FUNCTION_BLOCK Automatik_Betrieb
VAR_INPUT
	Kein_Notaus : BOOL;
	Zyklus_Start : BOOL;
	Zyklus_Stopp : BOOL;
	SFCInit : BOOL;
	SFCTip : BOOL;
	SFCTipMode : BOOL;
	Einfache_Klemmung : BOOL;
	
	//Eingänge Sensorik
	//Zuführer
	Endl_Zufuehrer_Hinten : BOOL;
	Endl_Zufuehrer_Vorne : BOOL;
	Vorposition_Zufuehrer : BOOL;
	IOL_Schaltausg_Distanzsensor_Holzende : BOOL; //Über Schaltausgang oder IO-Link Analogdaten?
	IOL_DistanzSensor_Abst : UINT;
	//Stammklemmung Oben
	Endl_Obere_Stammklemmung_Oben : BOOL;
	Endl_Obere_Stammklemmung_Unten : BOOL;
	Endl_Tastschiene : BOOL;
	Schaltausg_Druckschalter_Obere_Klemmung : BOOL;
	//Stammklemmung Unten
	Endl_Untere_Stammklemmung_Oben : BOOL;
	Endl_Untere_Stammklemmung_Unten : BOOL;
	//Säge
	Endl_Saege_Oben : BOOL;
	Endl_Saege_Unten : BOOL;
	
END_VAR
VAR_OUTPUT
	Warten_Auf_Weiterschalten :BOOL;
	Warten_auf_Material : BOOL;
	//Hydraulik
	QStammklemmung_Oben_Hoch : BOOL;
	QStammklemmung_Oben_Runter : BOOL;
	QStammklemmung_Unten_Hoch : BOOL;
	QStammklemmung_Unten_Runter : BOOL;
	QSaege_Senken : BOOL;
	QSaege_Heben : BOOL;
	//Ausgänge Schalten
	QHydraulikpumpe_EIN : BOOL;
	QZufuehrer_Antrieb_vor : BOOL;
	QZufuehrer_Antrieb_Rueck : BOOL;
	QSaege_Antrieb_Ein : BOOL;
	QKettenschmierung_EIN : BOOL;
	
END_VAR
VAR_IN_OUT
	warten : BOOL;
	Hydraulik_EIN : BOOL;
	Zyklus_Beendet : BOOL;
END_VAR
VAR
	Holz_Fertig : BOOL;
	Holz_Geklemmt : BOOL;
END_VAR

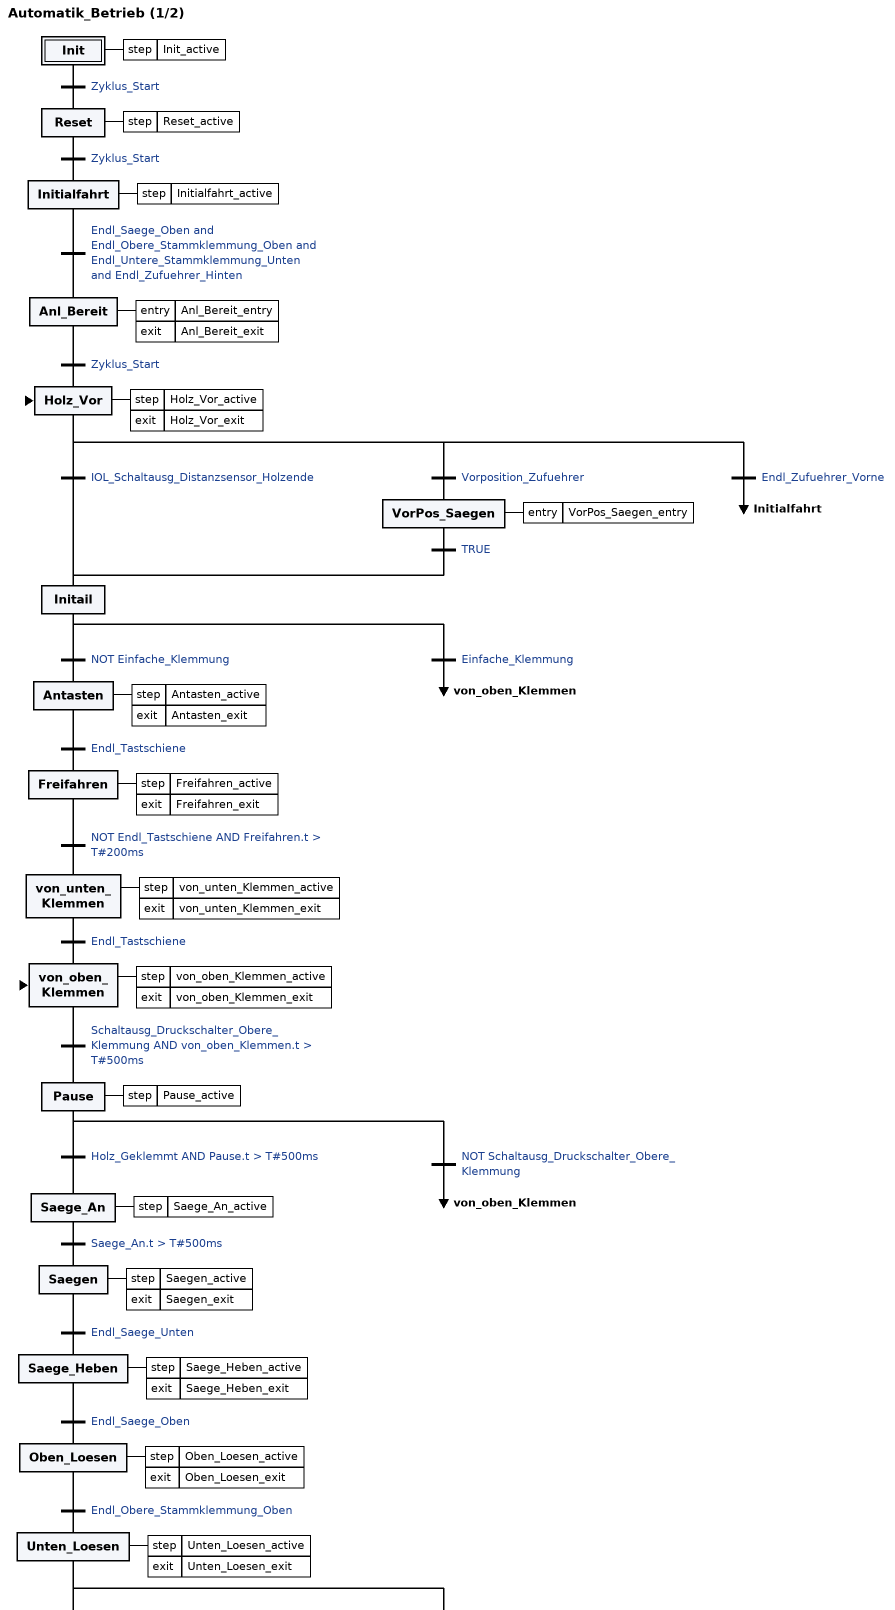
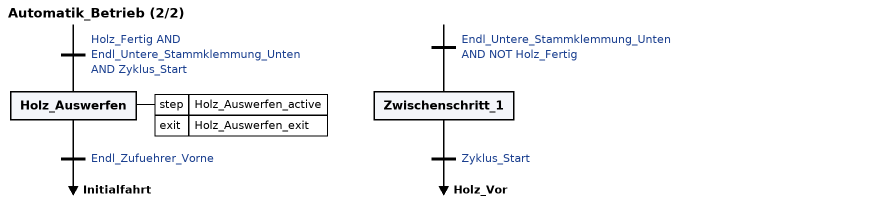
INITIAL_STEP Init:
    Init_active(N);  // step action
END_STEP
TRANSITION FROM Init TO Reset
    := Zyklus_Start;
END_TRANSITION
STEP Reset:
    Reset_active(N);  // step action
END_STEP
TRANSITION FROM Reset TO Initialfahrt_
    := Zyklus_Start;
END_TRANSITION
STEP Initialfahrt_:  // name as stored: Initialfahrt 
    Initialfahrt_active(N);  // step action
END_STEP
TRANSITION FROM Initialfahrt_ TO Anl_Bereit
    := Endl_Saege_Oben and Endl_Obere_Stammklemmung_Oben and Endl_Untere_Stammklemmung_Unten and Endl_Zufuehrer_Hinten;
END_TRANSITION
STEP Anl_Bereit:
    Anl_Bereit_entry(P1);  // entry action
    Anl_Bereit_exit(P0);  // exit action
END_STEP
TRANSITION FROM Anl_Bereit TO Holz_Vor
    := Zyklus_Start;
END_TRANSITION
STEP Holz_Vor:
    Holz_Vor_active(N);  // step action
    Holz_Vor_exit(P0);  // exit action
END_STEP
TRANSITION FROM Holz_Vor TO Initail
    := IOL_Schaltausg_Distanzsensor_Holzende;
END_TRANSITION
TRANSITION FROM Holz_Vor TO VorPos_Saegen
    := Vorposition_Zufuehrer;
END_TRANSITION
STEP VorPos_Saegen:
    VorPos_Saegen_entry(P1);  // entry action
END_STEP
TRANSITION FROM VorPos_Saegen TO Initail
    := TRUE;
END_TRANSITION
TRANSITION FROM Holz_Vor TO Initialfahrt
    := Endl_Zufuehrer_Vorne;
END_TRANSITION
// macro Holz_Klemmen begins
STEP Initail:
END_STEP
TRANSITION FROM Initail TO Antasten
    := NOT Einfache_Klemmung;
END_TRANSITION
STEP Antasten:
    Antasten_active(N);  // step action
    Antasten_exit(P0);  // exit action
END_STEP
TRANSITION FROM Initail TO von_oben_Klemmen
    := Einfache_Klemmung;
END_TRANSITION
TRANSITION FROM Antasten TO Freifahren
    := Endl_Tastschiene;
END_TRANSITION
STEP Freifahren:
    Freifahren_active(N);  // step action
    Freifahren_exit(P0);  // exit action
END_STEP
TRANSITION FROM Freifahren TO von_unten_Klemmen
    := NOT Endl_Tastschiene AND Freifahren.t > T#200ms;
END_TRANSITION
STEP von_unten_Klemmen:
    von_unten_Klemmen_active(N);  // step action
    von_unten_Klemmen_exit(P0);  // exit action
END_STEP
TRANSITION FROM von_unten_Klemmen TO von_oben_Klemmen
    := Endl_Tastschiene;
END_TRANSITION
STEP von_oben_Klemmen:
    von_oben_Klemmen_active(N);  // step action
    von_oben_Klemmen_exit(P0);  // exit action
END_STEP
TRANSITION FROM von_oben_Klemmen TO Pause
    := Schaltausg_Druckschalter_Obere_Klemmung AND von_oben_Klemmen.t > T#500ms;
END_TRANSITION
STEP Pause:
    Pause_active(N);  // step action
END_STEP
TRANSITION FROM Pause TO Saege_An
    := Holz_Geklemmt AND Pause.t > T#500ms;
END_TRANSITION
TRANSITION FROM Pause TO von_oben_Klemmen
    := NOT Schaltausg_Druckschalter_Obere_Klemmung;
END_TRANSITION
// macro Holz_Saegen begins
STEP Saege_An:
    Saege_An_active(N);  // step action
END_STEP
TRANSITION FROM Saege_An TO Saegen
    := Saege_An.t > T#500ms;
END_TRANSITION
STEP Saegen:
    Saegen_active(N);  // step action
    Saegen_exit(P0);  // exit action
END_STEP
TRANSITION FROM Saegen TO Saege_Heben
    := Endl_Saege_Unten;
END_TRANSITION
STEP Saege_Heben:
    Saege_Heben_active(N);  // step action
    Saege_Heben_exit(P0);  // exit action
END_STEP
TRANSITION FROM Saege_Heben TO Oben_Loesen
    := Endl_Saege_Oben;
END_TRANSITION
// macro Holz_Klemmung_Loesen begins
STEP Oben_Loesen:
    Oben_Loesen_active(N);  // step action
    Oben_Loesen_exit(P0);  // exit action
END_STEP
TRANSITION FROM Oben_Loesen TO Unten_Loesen
    := Endl_Obere_Stammklemmung_Oben;
END_TRANSITION
STEP Unten_Loesen:
    Unten_Loesen_active(N);  // step action
    Unten_Loesen_exit(P0);  // exit action
END_STEP
TRANSITION FROM Unten_Loesen TO Holz_Auswerfen
    := Holz_Fertig AND Endl_Untere_Stammklemmung_Unten AND Zyklus_Start;
END_TRANSITION
STEP Holz_Auswerfen:
    Holz_Auswerfen_active(N);  // step action
    Holz_Auswerfen_exit(P0);  // exit action
END_STEP
TRANSITION FROM Holz_Auswerfen TO Initialfahrt
    := Endl_Zufuehrer_Vorne;
END_TRANSITION
TRANSITION FROM Unten_Loesen TO Zwischenschritt_1
    := Endl_Untere_Stammklemmung_Unten AND NOT Holz_Fertig;
END_TRANSITION
STEP Zwischenschritt_1:
END_STEP
TRANSITION FROM Zwischenschritt_1 TO Holz_Vor
    := Zyklus_Start;
END_TRANSITION

ACTION Anl_Bereit_entry:
Warten_auf_Material := TRUE;
QHydraulikpumpe_EIN := FALSE;
END_ACTION

ACTION Anl_Bereit_exit:
Warten_auf_Material := FALSE;
QHydraulikpumpe_EIN := TRUE;
END_ACTION

ACTION Antasten_active:
QStammklemmung_Oben_Runter := TRUE;
END_ACTION

ACTION Antasten_exit:
QStammklemmung_Oben_Runter := FALSE;
END_ACTION

ACTION Freifahren_active:
QStammklemmung_Oben_Hoch := TRUE;
END_ACTION

ACTION Freifahren_exit:
QStammklemmung_Oben_Hoch := FALSE;
END_ACTION

ACTION Holz_Auswerfen_active:
QZufuehrer_Antrieb_vor := TRUE;
END_ACTION

ACTION Holz_Auswerfen_exit:
QZufuehrer_Antrieb_vor := FALSE;
Holz_Fertig := FALSE;
END_ACTION

ACTION Holz_Vor_active:
IF NOT Vorposition_Zufuehrer AND NOT Endl_Zufuehrer_Vorne THEN
	QZufuehrer_Antrieb_vor := TRUE;
END_IF 


IF Vorposition_Zufuehrer OR Endl_Zufuehrer_Vorne OR IOL_Schaltausg_Distanzsensor_Holzende THEN
	QZufuehrer_Antrieb_vor := FALSE;
END_IF
END_ACTION

ACTION Holz_Vor_exit:
QZufuehrer_Antrieb_vor := FALSE;
END_ACTION

ACTION Init_active:
QStammklemmung_Oben_Hoch := 
QStammklemmung_Oben_Runter := 
QStammklemmung_Unten_Hoch := 
QStammklemmung_Unten_Runter := 
QSaege_Senken := 
QSaege_Heben := 
//Ausgänge Schalten
QHydraulikpumpe_EIN := 
QZufuehrer_Antrieb_vor := 
QZufuehrer_Antrieb_Rueck := 
QSaege_Antrieb_Ein := 
QKettenschmierung_EIN := 
Warten_Auf_Weiterschalten :=
Zyklus_Beendet := FALSE;
END_ACTION

ACTION Initialfahrt_active:
IF NOT Endl_Saege_Oben THEN
	QSaege_Heben := TRUE;
	warten := TRUE;
ELSE 
	QSaege_Heben := FALSE;
	warten := FALSE;
END_IF

IF NOT Endl_Obere_Stammklemmung_Oben AND NOT warten THEN
	QStammklemmung_Oben_Hoch := TRUE;
	warten := TRUE;
ELSE
	QStammklemmung_Oben_Hoch := FALSE;
	warten := FALSE;
END_IF

IF NOT Endl_Untere_Stammklemmung_Unten AND NOT warten THEN 
	QStammklemmung_Unten_Runter := TRUE;
	warten := TRUE;
ELSE 
	QStammklemmung_Unten_Runter := FALSE;
	warten := FALSE;
END_IF

IF NOT Endl_Zufuehrer_Hinten THEN
	QZufuehrer_Antrieb_Rueck := TRUE;
ELSE 
	QZufuehrer_Antrieb_Rueck := FALSE;
END_IF
END_ACTION

ACTION Oben_Loesen_active:
QStammklemmung_Oben_Hoch := TRUE;
END_ACTION

ACTION Oben_Loesen_exit:
QStammklemmung_Oben_Hoch := FALSE;
END_ACTION

ACTION Pause_active:
Holz_Geklemmt := TRUE;
END_ACTION

ACTION Reset_active:
//Hydraulik
QStammklemmung_Oben_Hoch := 
QStammklemmung_Oben_Runter := 
QStammklemmung_Unten_Hoch := 
QStammklemmung_Unten_Runter := 
QSaege_Senken := 
QSaege_Heben := 
//Ausgänge Schalten
QHydraulikpumpe_EIN := 
QZufuehrer_Antrieb_vor := 
QZufuehrer_Antrieb_Rueck := 
QSaege_Antrieb_Ein := 
QKettenschmierung_EIN := 
Warten_Auf_Weiterschalten :=
Zyklus_Beendet := FALSE;

QHydraulikpumpe_EIN := TRUE;
END_ACTION

ACTION Saege_An_active:
QSaege_Antrieb_Ein := TRUE;
END_ACTION

ACTION Saege_Heben_active:
QSaege_Heben := TRUE;
END_ACTION

ACTION Saege_Heben_exit:
QSaege_Heben := FALSE;
QSaege_Antrieb_Ein := FALSE;
END_ACTION

ACTION Saegen_active:
QSaege_Senken := TRUE;
END_ACTION

ACTION Saegen_exit:
QSaege_Senken := FALSE;
END_ACTION

ACTION Unten_Loesen_active:
QStammklemmung_Unten_Runter := TRUE;
END_ACTION

ACTION Unten_Loesen_exit:
QStammklemmung_Unten_Runter := FALSE;
END_ACTION

ACTION von_oben_Klemmen_active:
QStammklemmung_Oben_Runter := TRUE;
END_ACTION

ACTION von_oben_Klemmen_exit:
QStammklemmung_Oben_Runter := FALSE;
END_ACTION

ACTION von_unten_Klemmen_active:
QStammklemmung_Unten_Hoch := TRUE;
END_ACTION

ACTION von_unten_Klemmen_exit:
QStammklemmung_Unten_Hoch := FALSE;
END_ACTION

ACTION VorPos_Saegen_entry:
Holz_Fertig := True;
END_ACTION

END_FUNCTION_BLOCK

(* stored: Version 1.1.0.1, ProductVersion 3.1.4024.16
   POU Automatik_Betrieb: Id {389c9999-3a59-4eae-a5d7-775f0832929f}, SpecialFunc None
   Action Anl_Bereit_entry: Id {e773d2be-07aa-4d92-b0f4-5643f324081a}
   Action Anl_Bereit_exit: Id {73cf0ee5-ec99-4c2a-a3b7-2130806987ae}
   Action Antasten_active: Id {9aeb3b24-da66-4503-b15b-0bf23e9d07a3}
   Action Antasten_exit: Id {e228e9e9-7f26-4154-9731-9316d98f68d6}
   Action Freifahren_active: Id {ee037f1a-1729-4ea6-9af9-31fd4d6cdc5c}
   Action Freifahren_exit: Id {d4c5b9c5-5d99-46a0-ae13-75a71ee60ea0}
   Action Holz_Auswerfen_active: Id {1a2d9e2d-4ed9-42ef-a9e8-38c5f81ceaf2}
   Action Holz_Auswerfen_exit: Id {1de60d9c-bc22-4eff-a9ab-d16a0ffaf0a2}
   Action Holz_Vor_active: Id {ae9c850e-dfd9-47d0-b81d-0a71babc98c5}
   Action Holz_Vor_exit: Id {e0530356-532e-40fa-90f1-88a067669b06}
   Action Init_active: Id {9345cd39-b6a8-4d8e-9a83-cf662bdae352}
   Action Initialfahrt_active: Id {3a592d82-235e-4e01-98bb-2a8a17d3bf23}
   Action Oben_Loesen_active: Id {63a82339-152f-40b3-a547-93adeee09f71}
   Action Oben_Loesen_exit: Id {8d488609-627d-4e2a-8399-9da08a9f6ac1}
   Action Pause_active: Id {00832697-5248-4af7-a8b0-3d5991131cd7}
   Action Reset_active: Id {655ea83a-bad9-42e6-8025-12d370509b5e}
   Action Saege_An_active: Id {926a8648-21ef-45aa-8667-2aca32b4168f}
   Action Saege_Heben_active: Id {2e0c349c-729f-4fe5-99bd-b291bf07b2ad}
   Action Saege_Heben_exit: Id {4f9c9dba-a86f-4e63-90aa-88dd12507fa0}
   Action Saegen_active: Id {e870bf57-2355-4ee1-830c-a110f1de3b90}
   Action Saegen_exit: Id {7f40bc59-8c03-4701-85c1-56ecc1293c2b}
   Action Unten_Loesen_active: Id {4ff0307f-62d3-4c2f-ab7a-da793821a2ae}
   Action Unten_Loesen_exit: Id {d824afb0-3491-4dd7-8b1f-d177084ea825}
   Action von_oben_Klemmen_active: Id {9622a9a7-06b3-4eea-a86b-5f1fbdcf62c1}
   Action von_oben_Klemmen_exit: Id {d4ab5da3-b9ad-4e42-8da2-3598a9e9fdff}
   Action von_unten_Klemmen_active: Id {80206357-8cba-4cd7-b1c4-5bdb48a4dfea}
   Action von_unten_Klemmen_exit: Id {1c6a7bb6-a9c1-4b07-beb4-c5de9d459076}
   Action VorPos_Saegen_entry: Id {fa01a4c2-32ab-4762-9461-a2d314914d38} *)
